// TIA Portal V18 export
VAR_GLOBAL   // PLC tag table "Marking"
END_VAR
VAR_GLOBAL CONSTANT   // user constants
   MODE_LASER_MARKING_IDLE : Int := 0;
   MODE_LASER_MARKING_START : Int := 1;
   MODE_LASER_MARKING_WRITE : Int := 2;
   MODE_LASER_MARKING_WRITE_ALL : Int := 3;
   MODE_LASER_MARKING_READ_CODE : Int := 4;
END_VAR
